# EPICS substitutions: keithley2000ScanApp/Db/keithley2000ScanChannel.substitutions
file "db/keithley2000ScanChannel.template"
{
pattern
{INDEX}
{"A"}
{"B"}
}
